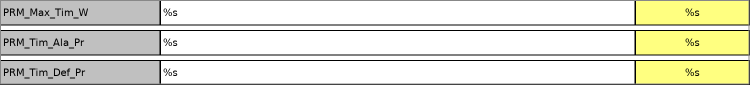
VISUALIZATION VISU_CONFIG_VANNE_ASS_VVAT653_ETHERCAT  // 750x85
(*visualistion pour secondaire dans chambre et primaire dans sas ==> paramètres pour chambre*)
VAR_IN_OUT
	m_Input_Vanne : BLOCK_VVAT_653_ETHERCAT;
END_VAR
    Rectangle (160,0 475x25), "%s", text list: 'TextList_VVAT_650_ETHERCAT', text index: 1
    Rectangle (635,0 115x25), "%s", text variable: m_Input_Vanne.PRM_Max_Tim_W, input disabled if: NOT Global_Variables.PRG_USER.ACTU_USER.CONF_MACHINE
        OnMouseClick: write the text variable via InputWithLimits
    Rectangle (0,0 160x25), "PRM_Max_Tim_W"
    Rectangle (160,30 475x25), "%s", text list: 'TextList_VVAT_650_ETHERCAT', text index: 2
    Rectangle (635,30 115x25), "%s", text variable: m_Input_Vanne.PRM_Tim_Ala_Pr, input disabled if: NOT Global_Variables.PRG_USER.ACTU_USER.CONF_MACHINE
        OnMouseClick: write the text variable via InputWithLimits
    Rectangle (0,30 160x25), "PRM_Tim_Ala_Pr"
    Rectangle (0,60 160x25), "PRM_Tim_Def_Pr"
    Rectangle (160,60 475x25), "%s", text list: 'TextList_VVAT_650_ETHERCAT', text index: 3
    Rectangle (635,60 115x25), "%s", text variable: m_Input_Vanne.PRM_Tim_Def_Pr, input disabled if: NOT Global_Variables.PRG_USER.ACTU_USER.CONF_MACHINE
        OnMouseClick: write the text variable via InputWithLimits
END_VISUALIZATION

(* stored: Version 1.1.0.1, ProductVersion 3.1.4024.12
   Visu VISU_CONFIG_VANNE_ASS_VVAT653_ETHERCAT: Id {dfddcc0a-db3d-4279-b3a3-60397eb8636f} *)
